Fanuc KAREL source: kt00162.KL

-- PROVISIONAL review KL for V1013-1; original PC SHA256 ee647b4b4c94674d03f58e79ef9811f5e358a3b6f496f18e6df5a1fa3c998045
-- Incomplete behavior may be omitted. Consult companion uncertainty JSON. Do not deploy.
PROGRAM KT00162
%NOLOCKGROUP
VAR
  I1 : INTEGER
  I2 : INTEGER
  OUT : REAL
BEGIN
  -- UNRESOLVED_PC offsets 5-16; opcodes 2E,23
  -- UNRESOLVED_PC offsets 21-32; opcodes 2E,23
  -- UNRESOLVED_PC offsets 37-48; opcodes 2E,23
  -- UNRESOLVED_PC offsets 53-64; opcodes 2E,23
  -- UNRESOLVED_PC offsets 69-89; opcodes 21,21,56,64,23
  -- UNRESOLVED_PC offsets 94-98; opcodes 7F
END KT00162
